// Type alias for represeting position.
TYPE T_Position : LINT; END_TYPE

(* stored: Version 1.1.0.1
   DUT T_Position: Id {d0b68156-c1bb-0d16-286e-24e439888fe3} *)
